// TIA Portal V19 export
FUNCTION_BLOCK "TYPIC_C406_BF_CAD"   // FB10, FBD
TITLE = TYPIC_C406_BF_CAD: CaDo Tunnel
{ S7_Optimized_Access := 'TRUE' }
AUTHOR : OCOTECH
FAMILY : Typical
NAME : C406.801
// Logisch Object Besturing: C406.801
// 
// Het doel van de BF CAD (CaDo Tunnel) is om de algemene sturing te voorzien van de calamiteiten doorsteek.
// 
// De algemene sturing omvat het weergeven van de algemene toestand en het openen en sluiten van calamiteiten doorsteek ten behoeve van de hulpdiensten en werkverkeer.
// stored: MemoryReserve 10, SetENOAutomatically false
   VAR_INPUT
      STU_AUT_CMD { ExternalAccessible := 'False'; ExternalVisible := 'False'; ExternalWritable := 'False'} : USInt;   // Sturing calamiteitendoorsteek algemeen
      STU_ALG_LCK_SIG { ExternalAccessible := 'False'; ExternalVisible := 'False'; ExternalWritable := 'False'} : USInt;   // Onderdruk alarmen
      STU_CAD_LCK_SIG { ExternalAccessible := 'False'; ExternalVisible := 'False'; ExternalWritable := 'False'} : USInt;   // Onderdruk alarm Cado niet dicht
      CFG_TST_UTYD { ExternalAccessible := 'False'; ExternalVisible := 'False'; ExternalWritable := 'False'} : Time;   // Maximale transitietijd stand verandering calamiteitendoorsteek (transitiestatus niet bereikt)
      CFG_TST_OK_TYD { ExternalAccessible := 'False'; ExternalVisible := 'False'; ExternalWritable := 'False'} : Time;   // Stabilisatietijd voor de toestand OK (bereikt)
   END_VAR
   VAR_OUTPUT
      STU_CAD_CMD { ExternalAccessible := 'False'; ExternalVisible := 'False'; ExternalWritable := 'False'} : USInt;   // Sturing CaDo algemeen
   END_VAR
   VAR_IN_OUT
      VAR_CAD : Array[0..1] of Bool;   // Array met alle calamiteitendoorsteken, met alle variabelen van de calamiteitendoorsteek
   END_VAR
   VAR
      BED : Struct   // Bedieningen
         ALG : Struct   // Gewenste stand
            X : "UDT_BED_ALG";
            KNOP { S7_SetPoint := 'True'} : Array[0..3] of "UDT_BED_KNOP";
         END_STRUCT;
      END_STRUCT;
      BED_ALG { ExternalWritable := 'False'} : "TYPIC_HF_BED_ALG_KNOP";   // Gewenste stand
      SIG { ExternalWritable := 'False'} : Struct   // Signaleringen
         AA01 : Bool;   // Gewenste stand niet bereikt
         AB01 : Bool;   // CaDo niet beschikbaar
         AB02 : Bool;   // CaDo beperkt beschikbaar
         AV01 : Bool;   // CaDo niet dicht
      END_STRUCT;
      VAR { ExternalWritable := 'False'} : Struct   // Variabelen
         BMO : USInt;   // Bedieningsmode
         TST_BWA : USInt;   // De status van de transitie van de CaDo
         BSC : USInt;   // Geeft de beschikbaarheidsstatus van de CaDo aan
         CAD_SWA : USInt;   // Doelstand CaDo
         CAD_BWA : USInt;   // Werkelijke stand CaDo
         VGV_SIG_VOP : Bool;   // TRUE = Signaleringen vrijgegeven voor verkeersoperator FALSE = Onderdrukt
      END_STRUCT;
      HF_TST { ExternalAccessible := 'False'; ExternalVisible := 'False'; ExternalWritable := 'False'} : "TYPIC_HF_TST";   // Hulpfunctie transitiestatus
   END_VAR
   // // BED.ALG.KNOP[0] : Auto
   // // BED.ALG.KNOP[1] : Open
   // // BED.ALG.KNOP[2] : Dicht
   // // BED.ALG.KNOP[3] : Stop
BEGIN

REGION Network 1: START
END_REGION

REGION Network 2: +++ Bedieningen +++
   // Vrijgave en verwerking van de bedieningen (centrale en lokale bediening). De bedienwaardes worden daarna in de verdere deelfunctionaliteiten gebruikt.
END_REGION

REGION Network 3: Knoppen BED_ALG(Gewenste stand)
   // Waardes en vrijge van de knoppen BED_ALG
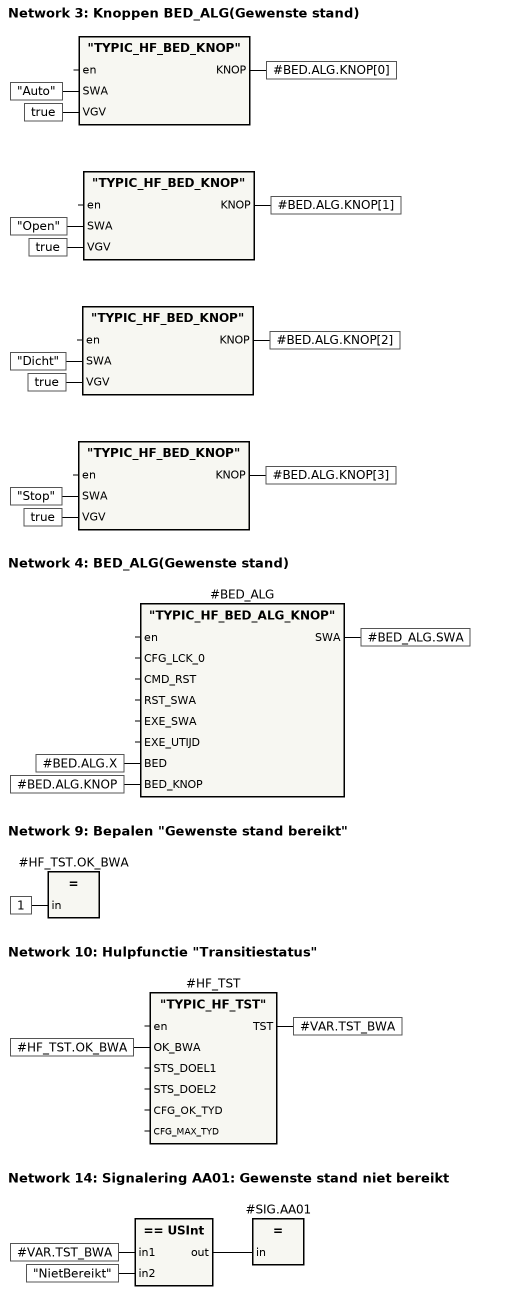
   "TYPIC_HF_BED_KNOP"(SWA := "Auto", VGV := true, KNOP => #BED.ALG.KNOP[0]);
   "TYPIC_HF_BED_KNOP"(SWA := "Open", VGV := true, KNOP => #BED.ALG.KNOP[1]);
   "TYPIC_HF_BED_KNOP"(SWA := "Dicht", VGV := true, KNOP => #BED.ALG.KNOP[2]);
   "TYPIC_HF_BED_KNOP"(SWA := "Stop", VGV := true, KNOP => #BED.ALG.KNOP[3]);
END_REGION

REGION Network 4: BED_ALG(Gewenste stand)
   // Verwerking BED_ALG
   #BED_ALG(BED := #BED.ALG.X, BED_KNOP := #BED.ALG.KNOP, SWA => #BED_ALG.SWA);   // "TYPIC_HF_BED_ALG_KNOP"
END_REGION

REGION Network 5: +++ Bedieningsmode +++
   // Bedieningsmode (Auto / Manueel ) bepalen.
END_REGION

REGION Network 6: +++ Bepalen gewenst stand +++
   // Bepalen van de gewenste stand (Open / Dicht / Stop)
END_REGION

REGION Network 7: +++ Bepalen werkelijke stand +++
   // Bepalen van de werkelijke stand (Open / Dicht / DichtVerlaten / Onbepaald) aan de hand van positiestatus van de calamiteitendoorsteken.
END_REGION

REGION Network 8: +++ Bepalen transitiestatus +++
   // Transitiestatus (bereikt / niet bereikt / in transitie) bepalen.
END_REGION

REGION Network 9: Bepalen "Gewenste stand bereikt"
   // Bepalen of de actuele stand in overeenstemming is met de gewenste stand
   #HF_TST.OK_BWA := 1;
END_REGION

REGION Network 10: Hulpfunctie "Transitiestatus"
   // De transitiestatus geeft de relatie tussen een gewenste stand (van een functionaliteit) en de actuele stand aan.
   #HF_TST(OK_BWA := #HF_TST.OK_BWA, TST => #VAR.TST_BWA);   // "TYPIC_HF_TST"
END_REGION

REGION Network 11: +++ Bepalen beschikbaarheidsstatus +++
   // Beschikbaarheidsstatus (beschikbaar / beperkt beschikbaar / niet beschikbaar) bepalen.
END_REGION

REGION Network 12 (SCL): Beschikbaarheidsstatus bepalen
   IF 
       //voorwaarden "Niet beschikbaar"
       TRUE
   THEN
       //Beschikbaarheidsstatus = Niet Beschikbaar
       #VAR.BSC:= "NietBeschikbaar";
   ELSIF
       //voorwaarden "Beperkt beschikbaar"
       TRUE
   THEN
       //Beschikbaarheidsstatus = Beperkt Beschikbaar
       #VAR.BSC:= "Beperkt";
   ELSE
       //Beschikbaarheidsstatus = Beschikbaar
       #VAR.BSC:= "Beschikbaar";
   END_IF;
END_REGION

REGION Network 13: +++ Signaleringen +++
   // Aanmaken signaleringen.
END_REGION

REGION Network 14: Signalering AA01: Gewenste stand niet bereikt
   #SIG.AA01 := #VAR.TST_BWA = "NietBereikt";
END_REGION

REGION Network 15: Signalering AB01 : Niet Beschikbaar
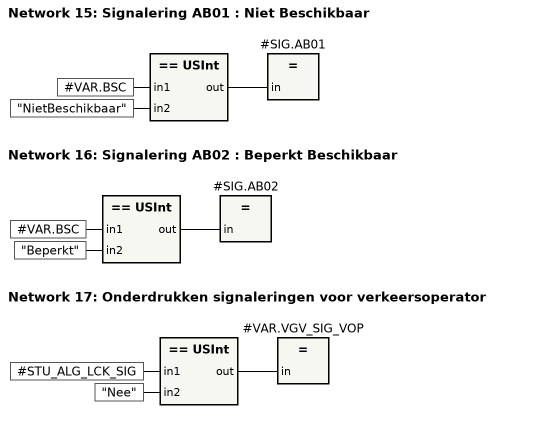
   #SIG.AB01 := #VAR.BSC = "NietBeschikbaar";
END_REGION

REGION Network 16: Signalering AB02 : Beperkt Beschikbaar
   #SIG.AB02 := #VAR.BSC = "Beperkt";
END_REGION

REGION Network 17: Onderdrukken signaleringen voor verkeersoperator
   // Via de variabele VGV_SIG_VOP wordt aan IRIS SCADA doorgegeven of signaleringen (bestemd voor de verkeersoperator) van de deze functie zichtbaar (of onderdrukt) moeten zijn.
   #VAR.VGV_SIG_VOP := #STU_ALG_LCK_SIG = "Nee";
END_REGION

REGION Network 18: +++ Sturingen +++
   // Individuele commandos uitsturen naar iedere calamiteiten doorsteek om te openen en te sluiten.
END_REGION

REGION Network 19: EINDE
   // Variabelen van intern scada rakvlak naar outputs copieren
END_REGION
END_FUNCTION_BLOCK
